FUNCTION ASSEMBLE_DWORD_FROM_BOOLS (* this Function combines the 32 BOOLS to a DWORD *)
  (* Standard: 61499-1; Description: Copyright (c) 2024 HR Agrartechnik GmbH This program and the accompanying materials are made available under the terms of the Eclipse Public License 2.0 which is available at https://www.eclipse.org/legal/epl-2.0/ SPDX-License-Identifier: EPL-2.0 *)
  (* Version 1.0, 2024-02-22, Franz H??pfinger, HR Agrartechnik, initial Implementation *)
  (* Version 1.1, 2024-07-28, Moritz Ortmeier, HR Agrartechnik, rename Function and change Input/Output Variables *)
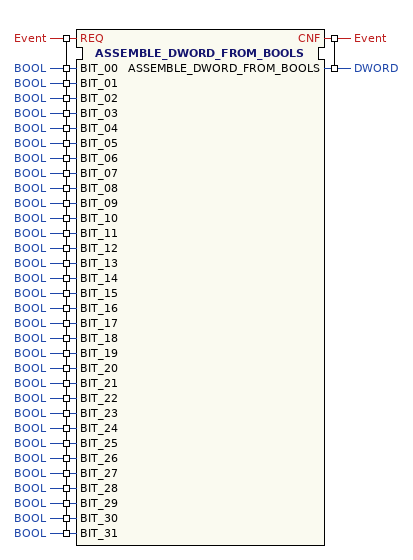
  EVENT_INPUT
    REQ WITH BIT_00, BIT_01, BIT_02, BIT_03, BIT_04, BIT_05, BIT_06, BIT_07, BIT_08, BIT_09, BIT_10, BIT_11, BIT_12, BIT_13, BIT_14, BIT_15, BIT_16, BIT_17, BIT_18, BIT_19, BIT_20, BIT_21, BIT_22, BIT_23, BIT_24, BIT_25, BIT_26, BIT_27, BIT_28, BIT_29, BIT_30, BIT_31;
  END_EVENT
  EVENT_OUTPUT
    CNF WITH ASSEMBLE_DWORD_FROM_BOOLS;
  END_EVENT
  VAR_INPUT
    BIT_00 : BOOL;
    BIT_01 : BOOL;
    BIT_02 : BOOL;
    BIT_03 : BOOL;
    BIT_04 : BOOL;
    BIT_05 : BOOL;
    BIT_06 : BOOL;
    BIT_07 : BOOL;
    BIT_08 : BOOL;
    BIT_09 : BOOL;
    BIT_10 : BOOL;
    BIT_11 : BOOL;
    BIT_12 : BOOL;
    BIT_13 : BOOL;
    BIT_14 : BOOL;
    BIT_15 : BOOL;
    BIT_16 : BOOL;
    BIT_17 : BOOL;
    BIT_18 : BOOL;
    BIT_19 : BOOL;
    BIT_20 : BOOL;
    BIT_21 : BOOL;
    BIT_22 : BOOL;
    BIT_23 : BOOL;
    BIT_24 : BOOL;
    BIT_25 : BOOL;
    BIT_26 : BOOL;
    BIT_27 : BOOL;
    BIT_28 : BOOL;
    BIT_29 : BOOL;
    BIT_30 : BOOL;
    BIT_31 : BOOL;
  END_VAR
  VAR_OUTPUT
    ASSEMBLE_DWORD_FROM_BOOLS : DWORD;
  END_VAR
  BODY IN ST:
(* this Function combines the 32 BOOLS to a DWORD *)
FUNCTION ASSEMBLE_DWORD_FROM_BOOLS : DWORD

VAR_INPUT
	BIT_00 : BOOL;
	BIT_01 : BOOL;
	BIT_02 : BOOL;
	BIT_03 : BOOL;
	BIT_04 : BOOL;
	BIT_05 : BOOL;
	BIT_06 : BOOL;
	BIT_07 : BOOL;
	BIT_08 : BOOL;
	BIT_09 : BOOL;
	BIT_10 : BOOL;
	BIT_11 : BOOL;
	BIT_12 : BOOL;
	BIT_13 : BOOL;
	BIT_14 : BOOL;
	BIT_15 : BOOL;
	BIT_16 : BOOL;
	BIT_17 : BOOL;
	BIT_18 : BOOL;
	BIT_19 : BOOL;
	BIT_20 : BOOL;
	BIT_21 : BOOL;
	BIT_22 : BOOL;
	BIT_23 : BOOL;
	BIT_24 : BOOL;
	BIT_25 : BOOL;
	BIT_26 : BOOL;
	BIT_27 : BOOL;
	BIT_28 : BOOL;
	BIT_29 : BOOL;
	BIT_30 : BOOL;
	BIT_31 : BOOL;
END_VAR

ASSEMBLE_DWORD_FROM_BOOLS.%X0 := BIT_00;
ASSEMBLE_DWORD_FROM_BOOLS.%X1 := BIT_01;
ASSEMBLE_DWORD_FROM_BOOLS.%X2 := BIT_02;
ASSEMBLE_DWORD_FROM_BOOLS.%X3 := BIT_03;
ASSEMBLE_DWORD_FROM_BOOLS.%X4 := BIT_04;
ASSEMBLE_DWORD_FROM_BOOLS.%X5 := BIT_05;
ASSEMBLE_DWORD_FROM_BOOLS.%X6 := BIT_06;
ASSEMBLE_DWORD_FROM_BOOLS.%X7 := BIT_07;
ASSEMBLE_DWORD_FROM_BOOLS.%X8 := BIT_08;
ASSEMBLE_DWORD_FROM_BOOLS.%X9 := BIT_09;
ASSEMBLE_DWORD_FROM_BOOLS.%X10 := BIT_10;
ASSEMBLE_DWORD_FROM_BOOLS.%X11 := BIT_11;
ASSEMBLE_DWORD_FROM_BOOLS.%X12 := BIT_12;
ASSEMBLE_DWORD_FROM_BOOLS.%X13 := BIT_13;
ASSEMBLE_DWORD_FROM_BOOLS.%X14 := BIT_14;
ASSEMBLE_DWORD_FROM_BOOLS.%X15 := BIT_15;
ASSEMBLE_DWORD_FROM_BOOLS.%X16 := BIT_16;
ASSEMBLE_DWORD_FROM_BOOLS.%X17 := BIT_17;
ASSEMBLE_DWORD_FROM_BOOLS.%X18 := BIT_18;
ASSEMBLE_DWORD_FROM_BOOLS.%X19 := BIT_19;
ASSEMBLE_DWORD_FROM_BOOLS.%X20 := BIT_20;
ASSEMBLE_DWORD_FROM_BOOLS.%X21 := BIT_21;
ASSEMBLE_DWORD_FROM_BOOLS.%X22 := BIT_22;
ASSEMBLE_DWORD_FROM_BOOLS.%X23 := BIT_23;
ASSEMBLE_DWORD_FROM_BOOLS.%X24 := BIT_24;
ASSEMBLE_DWORD_FROM_BOOLS.%X25 := BIT_25;
ASSEMBLE_DWORD_FROM_BOOLS.%X26 := BIT_26;
ASSEMBLE_DWORD_FROM_BOOLS.%X27 := BIT_27;
ASSEMBLE_DWORD_FROM_BOOLS.%X28 := BIT_28;
ASSEMBLE_DWORD_FROM_BOOLS.%X29 := BIT_29;
ASSEMBLE_DWORD_FROM_BOOLS.%X30 := BIT_30;
ASSEMBLE_DWORD_FROM_BOOLS.%X31 := BIT_31;
END_FUNCTION
  END_BODY
END_FUNCTION
